// TwinCAT 3 PLC project main
// ProgramVersion: 3.1.4024.0
// libraries:
//   Tc2_Standard, * (Beckhoff Automation GmbH)
//   Tc2_System, * (Beckhoff Automation GmbH)
//   Tc3_Module, * (Beckhoff Automation GmbH)
// project tree:
//   / GlobalTextList.TcGTLO, PlcTask.TcTTO, Visualization Manager.TcVMO (not stored)
//   POUs/ MAIN.TcPOU
//   VISUs/ Visu.TcVIS
// real-time tasks:
//   TASK PlcTask: cycle T#10ms, priority 20, ADS port 350

CONFIGURATION main
    RESOURCE PLC ON TwinCAT3
        TASK PlcTask(INTERVAL := T#10ms, PRIORITY := 20);
        PROGRAM MAIN WITH PlcTask : MAIN;
    END_RESOURCE
END_CONFIGURATION

// ---- POUs/MAIN.TcPOU
PROGRAM MAIN
VAR
	nPmeter AT %I* : INT;
	nScaledMax AT %Q* : INT := 15;
	nValue AT %Q* : INT;
END_VAR

//Lees de potentiometer in en verschaal deze waarden naar een getal tussen 0 en de variable nScaledMax. Geef voorlopig de initial value van 10 mee.

nValue := REAL_TO_BYTE(nPmeter/32767.0 * nScaledMax);

END_PROGRAM

// ---- VISUs/Visu.TcVIS
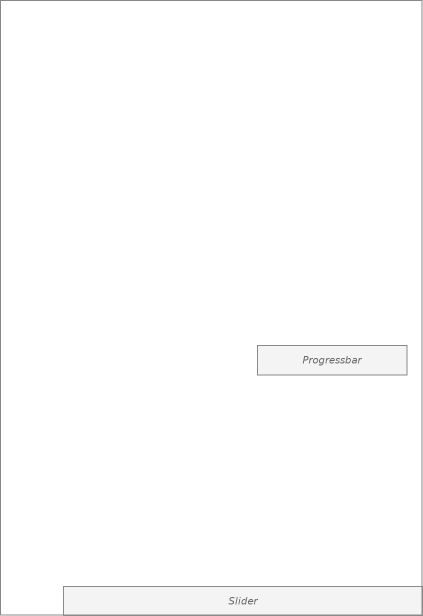
VISUALIZATION Visu  // 423x616
    Slider (63,586 360x30), variable: MAIN.nPmeter, scale 0..32767
    Progressbar (257,345 150x30), variable: MAIN.nValue
END_VISUALIZATION
